FUNCTION_BLOCK TcoTixonPickStep_v_1_x_x EXTENDS TcoCore.TcoComponent

VAR_INPUT
	inControllerInAuto  : BOOL;
	inNotEmptyFeeder  : BOOL;	
	inSeparatorHomePos  : BOOL;
	inFillingSensor  : BOOL; 
	inSeparatorPresent  : BOOL;
	inStepperHomePos  : BOOL;
	inStepperWorkPos  : BOOL;
	inSeparatorWorkPos  : BOOL;
END_VAR
VAR_OUTPUT
	outFeedingA : BOOL;
	outSepareComponent : BOOL;
	outBlowValveA : BOOL;
	outRedLed : BOOL;	
	outGreenLed : BOOL;
	outHopper : BOOL;
	outStepperValve : BOOL;
END_VAR
VAR

    {attribute addProperty Name "<#Status#>"}
    {attribute clr [ReadOnly()]}
    _status : TcoTixonPickStep_Status_v_1_x_x;
    {attribute addProperty Name "<#Control#>"}
    _control : TcoTixonPickStep_Control_v_1_x_x;
    {attribute addProperty Name "<#Config#>"}
    _config : TcoTixonPickStep_Config_v_1_x_x;

    _someTaskIsActive : BOOL;

    {attribute 'hide'}
    _blink : TcoUtilities.TcoBlinker(THIS^);
    _runAutomatic : BOOL;
    _hasError : BOOL;
END_VAR
VAR

    {attribute addProperty Name "<#Separator task#>"}
    _separatorTask : TcoTixonPickStepSeparatorTask(THIS^);
    {attribute addProperty Name "<#Buffer task#>"}
    _bufferTask : TcoTixonBufferTask(THIS^);
  	{attribute addProperty Name "<#Step task#>"}
    _stepperTask : TcoTixonPickStepTask(THIS^);
    {attribute addProperty Name "<#Hopper task#>"}
    _hopperTask : TcoTixonHopperTask(THIS^);

    {attribute addProperty Name "<#Restore#>"}
    _restoreTask : TcoCore.TcoTask(THIS^);

END_VAR

VAR
    {attribute 'hide'}
    _sb : TcoCore.StringBuilder;
END_VAR



_blink(inOnTime:=_config.BlinkTime,inOffTime:=_config.BlinkTime);		
UpdateStatus();

_separatorTask.Enabled:=TRUE;
_separatorTask(inoConfig:=_config,inoControl:=_control,inoStatus:=_status);
_bufferTask.Enabled:=TRUE;
_bufferTask(inoConfig:=_config,inoControl:=_control,inoStatus:=_status);
_stepperTask.Enabled:=TRUE;
_stepperTask(inoConfig:=_config,inoControl:=_control,inoStatus:=_status);
_hopperTask.Enabled := _config.HopperActive;
_hopperTask(inoConfig:=_config,inoControl:=_control,inoStatus:=_status);







//*************RESTORE********************

_restoreTask.Enabled := TRUE;
IF _restoreTask.Execute() THEN
	Restore();
	_restoreTask.DoneWhen(TRUE);
END_IF
//****************************************



//IF(_status.State.Error) THEN Messenger.Error(_sb.Clear().Append('<#Drive error no #>').Append(UDINT_TO_STRING(_status.State.EventId)).Append(' |[[0]AdvancedDiagnosticMessage]|').Append('.').Append('For details see the service mode').ToString()); END_IF;


UpdateControl();

METHOD PUBLIC BufferFeed : TcoCore.ITcoTaskStatus
BufferFeed:=_bufferTask.Invoke();
_bufferTask.AutoRestore:=false;
END_METHOD

(*~
	<docu>
		<summary>
			Gets the configuration of the Tixon PickStep. 					
		</summary>			
	</docu>	
~*)
PROPERTY Config : REFERENCE TO TcoTixonPickStep_Config_v_1_x_x
GET
Config REF= _config;
END_GET
END_PROPERTY

METHOD PUBLIC CyclicBufferFeed : TcoCore.ITcoTaskStatus
CyclicBufferFeed:=_bufferTask.Invoke();
_bufferTask.AutoRestore:=true;
END_METHOD

METHOD PUBLIC CyclicHopperFeed : TcoCore.ITcoTaskStatus
CyclicHopperFeed:=_hopperTask.Invoke();
_hopperTask.AutoRestore:=TRUE;
END_METHOD

METHOD PUBLIC CyclicSepare : TcoCore.ITcoTaskStatus
CyclicSepare:=_separatorTask.Invoke();
_separatorTask.AutoRestore:=true;
END_METHOD

METHOD PUBLIC CyclicStepperFeed : TcoCore.ITcoTaskStatus
VAR_INPUT
END_VAR
CyclicStepperFeed:=_stepperTask.Invoke();
_stepperTask.AutoRestore:=true;
END_METHOD

METHOD PUBLIC DefaultSignalisation
VAR_INPUT
END_VAR
// led signalisation
_hasError:=_separatorTask.Error OR _stepperTask.Error OR _bufferTask.Error;
_control.GreenLed:=FALSE;
_control.RedLed:=FALSE;
IF _blink.IsOn AND NOT _status.ControllerInAuto  THEN
	_control.GreenLed:=TRUE;
	_control.RedLed:=TRUE;
ELSIF _status.ControllerInAuto AND  _status.NotEmptyFeeder THEN
	_control.GreenLed:=TRUE;
ELSIF _blink.IsOn AND _status.ControllerInAuto AND NOT _status.NotEmptyFeeder THEN
	_control.RedLed:=TRUE;
END_IF
END_METHOD

METHOD PUBLIC HopperFeed : TcoCore.ITcoTaskStatus
HopperFeed:=_hopperTask.Invoke();
_hopperTask.AutoRestore:=false;
END_METHOD

(*~
	<docu>
		<summary>
			Restores this instance to the Ready state. Can be called explicitly or from within one of the restore mechanisms.	
		</summary>			
	</docu>	
~*)
METHOD Restore : ITcoRestorable
RestoreTasks();
_control.BlowAValve:=FALSE;
_control.FeedingA:=FALSE;
_control.GreenLed:=FALSE;
_control.RedLed:=FALSE;
_control.SepareComponent:=FALSE;
_control.StepperValve:=FALSE;
_control.Hooper:=FALSE;
END_METHOD

METHOD INTERNAL RestoreTasks
//_resetTask.Restore();

_separatorTask.Restore();
_bufferTask.Restore();
_stepperTask.Restore();
_hopperTask.Restore();
END_METHOD

METHOD PUBLIC Separe : TcoCore.ITcoTaskStatus
Separe:=_separatorTask.Invoke();
_separatorTask.AutoRestore:=false;
END_METHOD

(*~
	<docu>
		<summary>
		    Custom service (manual, maintenance) logic.
			This method must be implemented in derived class.
		</summary>			
	</docu>	
~*)
METHOD PROTECTED ServiceMode
END_METHOD

(*~
	<docu>
		<summary>
			Gets the status of the Tixon PickStep. 					
		</summary>			
	</docu>	
~*)
PROPERTY Status : REFERENCE TO TcoTixonPickStep_Status_v_1_x_x
GET
Status REF= _status;
END_GET
END_PROPERTY

METHOD PUBLIC StepperFeed : TcoCore.ITcoTaskStatus
VAR_INPUT
END_VAR
StepperFeed:=_stepperTask.Invoke();
_stepperTask.AutoRestore:=FALSE;
END_METHOD

METHOD INTERNAL UpdateControl
VAR_INPUT
END_VAR

VAR
	index: INT;
END_VAR
outBlowValveA:= _control.BlowAValve;
outFeedingA:=_control.FeedingA;
outGreenLed:=_control.GreenLed;
outRedLed:=_control.RedLed;
outSepareComponent:=_control.SepareComponent;
outStepperValve:=_control.StepperValve;

outHopper:=_control.Hooper;
END_METHOD

METHOD INTERNAL UpdateStatus
VAR
    
END_VAR
_status.NotEmptyFeeder:=inNotEmptyFeeder;
_status.FillingSensor:=inFillingSensor;
_status.SeparatorHomePos:=inSeparatorHomePos;
_status.SeparatorPresent:=inSeparatorPresent;
_status.SeparatorWorkPos:=inSeparatorWorkPos;
_status.ControllerInAuto:=inControllerInAuto;
END_METHOD

END_FUNCTION_BLOCK

(* stored: Version 1.1.0.1, ProductVersion 3.1.4024.12
   POU TcoTixonPickStep_v_1_x_x: Id {e2a69733-a4e2-0630-1c24-a72bf113d9f8}, SpecialFunc None
   Folder Operations: Id {1b1d1953-a52c-0707-3526-59b366ecfe72}
   Folder Loop: Id {17bce385-100a-0673-2a65-88d03d9edb6a}
   Folder Single: Id {ce68a6a1-6d0b-01bd-1aac-004c9ab5d412}
   Folder Task: Id {7bc9f2bf-5a7f-09bf-0f63-05dd45b33b28}
   Method BufferFeed: Id {23ad9cd4-2c4a-06b9-2f81-0dc350560127}
   Property Config: Id {175d044f-1652-0a17-2513-eb21bb7c4ca2}
   Get Get: Id {513e5df0-0be0-05bc-2bcb-929f4c388968}
   Method CyclicBufferFeed: Id {f360a9d6-abdd-01fe-0829-52bdcfbf9e5b}
   Method CyclicHopperFeed: Id {ea5c6767-f4ba-077c-1ba7-51ed300eb151}
   Method CyclicSepare: Id {a88f6f41-51f2-079a-3c86-91471faad6ca}
   Method CyclicStepperFeed: Id {b6968204-5251-07e0-0871-1857dab59a86}
   Method DefaultSignalisation: Id {9a55f639-006d-0abd-0f7e-cce8b420186f}
   Method HopperFeed: Id {1f499a0f-d09d-0d03-076a-cd20b75ad246}
   Method Restore: Id {9cf088e3-d91e-0f6f-3df8-ec09596724ad}
   Method RestoreTasks: Id {8555c1b2-737a-0076-2516-b3fce1659d55}
   Method Separe: Id {751db759-e6f9-0685-0767-2e3180999873}
   Method ServiceMode: Id {a62693d4-6faf-093d-3bbe-e8755502782a}
   Property Status: Id {d0ab0933-ec89-0854-1880-8573a9b64458}
   Get Get: Id {27592f22-bd39-086a-3670-599e047e4a05}
   Method StepperFeed: Id {6322714e-29e4-0cba-162b-ef1cadf2384d}
   Method UpdateControl: Id {d7832ece-df6c-067c-3144-c929cfec9ad6}
   Method UpdateStatus: Id {654f7ef3-39fc-0f42-3223-2db92b513c10} *)
